// TIA Portal V20 export
TYPE "LWONIK_typePackMLMode"
// stored: Access Published
   STRUCT
      production : Bool;
      maintanance : Bool;
      manual : Bool;
   END_STRUCT;
END_TYPE
